Yaskawa INFORM job: hydraulic_planes_program.JBI

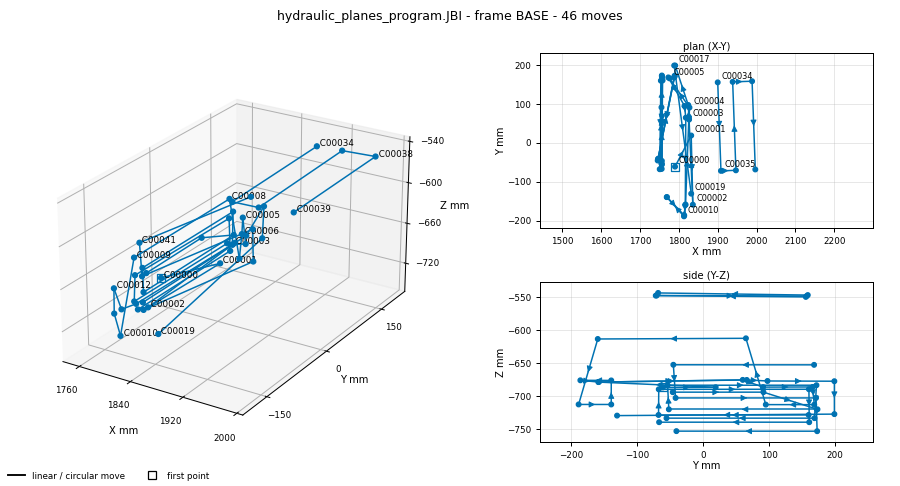
[picture p0: tool path of hydraulic_planes_program.JBI in frame BASE, 46 of 52 moves have a stored position in this frame; points joined in program order, loops and branches not executed]
/JOB
//NAME hydraulic_planes_program
//POS
///NPOS 46,0,46,0,0,0
///TOOL 0
///POSTYPE BASE
///RECTAN
///RCONF 0,0,0,0,0,0,0,0,0,0,0,0,0,0,0,0,0,0,0,0,0,0,0,0
C00000=1790.266260,-61.118146,-686.561623,175.000000,-86.957864,-5.000000
C00001=1831.954921,19.073830,-686.315651,175.000000,-89.878553,-42.967165
C00002=1836.147041,-158.971402,-678.483462,-5.000000,-59.939769,-144.273100
C00003=1826.434318,60.082030,-675.116712,5.000000,-61.318237,147.203233
C00004=1827.467674,91.039273,-686.093792,175.000000,-89.878553,-42.967165
C00005=1776.092305,166.200158,-685.860832,-175.000000,-89.999999,5.000000
C00006=1773.015262,168.636026,-712.737461,175.000000,-86.957864,-5.000000
C00007=1814.783866,95.105126,-712.668296,5.000000,-89.961663,134.868733
C00008=1817.982946,64.939100,-612.030081,175.000000,-59.162706,-36.238815
C00009=1816.677604,-159.909699,-613.050416,175.000000,-59.645373,36.364554
C00010=1813.343123,-188.991701,-712.402389,-175.000000,-89.962495,44.868708
C00011=1768.928091,-139.457958,-712.449114,-175.000000,-89.999999,5.000000
C00012=1769.441453,-139.453159,-675.944419,175.000000,-86.957864,-5.000000
C00013=1813.995933,-186.333152,-675.775252,175.000000,-89.860276,43.447212
C00014=1817.301672,-158.444384,-678.443506,175.000000,-60.142921,35.349719
C00015=1825.978625,66.227215,-675.229416,175.000000,-58.601867,-37.216727
C00016=1824.274715,97.685087,-676.791427,5.000000,-89.849901,133.447578
C00017=1790.762018,199.171368,-677.155686,-175.000000,-89.999999,5.000000
C00018=1788.152021,199.213725,-727.087548,175.000000,-86.957864,-5.000000
C00019=1831.944525,-130.625030,-729.338750,180.000000,-60.000000,0.000000
C00020=1756.349272,-46.141377,-693.754512,5.000000,-89.857180,175.000000
C00021=1755.399155,91.548361,-693.758382,5.000000,-89.857180,175.000000
C00022=1756.387865,173.552879,-719.824458,5.000000,-89.857180,175.000000
C00023=1755.391181,-52.033493,-719.824484,5.000000,-89.857180,175.000000
C00024=1755.768973,-53.986868,-683.221136,5.000000,-89.857180,175.000000
C00025=1756.321618,172.003597,-683.222222,5.000000,-89.857180,175.000000
C00026=1756.861736,169.068743,-733.220999,5.000000,-89.857180,175.000000
C00027=1756.478831,-55.593134,-733.219504,180.000000,-60.000000,0.000000
C00028=1753.816844,160.170606,-728.362357,-5.000000,-87.376565,175.000000
C00029=1750.864769,-67.689122,-728.388394,-5.000000,-87.376565,175.000000
C00030=1752.780642,-67.367991,-689.430064,-5.000000,-87.376565,175.000000
C00031=1756.818776,160.582398,-689.354311,-5.000000,-87.376565,175.000000
C00032=1758.269844,161.023273,-739.340500,-5.000000,-87.376565,175.000000
C00033=1755.987664,-66.800990,-739.335855,180.000000,-60.000000,0.000000
C00034=1900.141403,155.863057,-549.188650,175.000000,-5.000000,5.000000
C00035=1908.499765,-71.912467,-547.251638,175.000000,-5.000000,5.000000
C00036=1946.984303,-70.512261,-547.021638,175.000000,-5.000000,5.000000
C00037=1938.629923,157.154756,-547.865638,175.000000,-5.000000,5.000000
C00038=1988.606888,158.835908,-546.390638,175.000000,-5.000000,5.000000
C00039=1996.941331,-68.287794,-543.165638,175.000000,-5.000000,5.000000
C00040=1787.945105,168.400189,-652.296237,5.000000,-82.585527,-175.000000
C00041=1745.633077,-45.215626,-652.194331,5.000000,-82.585527,-175.000000
C00042=1746.401907,-41.803375,-702.518754,5.000000,-82.585527,-175.000000
C00043=1789.334500,171.346579,-702.527671,5.000000,-82.585527,-175.000000
C00044=1789.323694,173.045553,-753.012360,5.000000,-82.585527,-175.000000
C00045=1746.936745,-40.568483,-752.920252,180.000000,-60.000000,0.000000
///POSTYPE PULSE
///PULSE
EC00000=0.0
EC00001=0.0
EC00002=0.0
EC00003=0.0
EC00004=0.0
EC00005=0.0
EC00006=0.0
EC00007=0.0
EC00008=0.0
EC00009=0.0
EC00010=0.0
EC00011=0.0
EC00012=0.0
EC00013=0.0
EC00014=0.0
EC00015=0.0
EC00016=0.0
EC00017=0.0
EC00018=0.0
EC00019=0.0
EC00020=91136.0
EC00021=91136.0
EC00022=91136.0
EC00023=91136.0
EC00024=91136.0
EC00025=91136.0
EC00026=91136.0
EC00027=91136.0
EC00028=183296.0
EC00029=183296.0
EC00030=183296.0
EC00031=183296.0
EC00032=183296.0
EC00033=183296.0
EC00034=186368.0
EC00035=186368.0
EC00036=186368.0
EC00037=186368.0
EC00038=186368.0
EC00039=186368.0
EC00040=252928.0
EC00041=252928.0
EC00042=252928.0
EC00043=252928.0
EC00044=252928.0
EC00045=252928.0
//INST
///DATE 2023/08/16 16:00
///ATTR SC,RW,RJ
////FRAME BASE
///GROUP1 RB1,ST1
NOP
MOVJ P009 EX000 VJ=15.00
MOVJ C00000 EC00000 VJ=15.0
CALL JOB:SPYON
MOVL C00001 EC00001 V=150.0
MOVL C00002 EC00002 V=150.0
MOVL C00003 EC00003 V=150.0
MOVL C00004 EC00004 V=150.0
MOVL C00005 EC00005 V=150.0
MOVL C00006 EC00006 V=150.0
MOVL C00007 EC00007 V=150.0
MOVL C00008 EC00008 V=150.0
MOVL C00009 EC00009 V=150.0
MOVL C00010 EC00010 V=150.0
MOVL C00011 EC00011 V=150.0
MOVL C00012 EC00012 V=150.0
MOVL C00013 EC00013 V=150.0
MOVL C00014 EC00014 V=150.0
MOVL C00015 EC00015 V=150.0
MOVL C00016 EC00016 V=150.0
MOVL C00017 EC00017 V=150.0
MOVL C00018 EC00018 V=150.0
MOVL C00019 EC00019 V=150.0
CALL JOB:SPYOF
MOVJ P009 VJ=15.00
MOVJ C00020 EC00020 VJ=15.0
CALL JOB:SPYON
MOVL C00021 EC00021 V=150.0
MOVL C00022 EC00022 V=150.0
MOVL C00023 EC00023 V=150.0
MOVL C00024 EC00024 V=150.0
MOVL C00025 EC00025 V=150.0
MOVL C00026 EC00026 V=150.0
MOVL C00027 EC00027 V=150.0
CALL JOB:SPYOF
MOVJ P009 VJ=15.00
MOVJ C00028 EC00028 VJ=15.0
CALL JOB:SPYON
MOVL C00029 EC00029 V=150.0
MOVL C00030 EC00030 V=150.0
MOVL C00031 EC00031 V=150.0
MOVL C00032 EC00032 V=150.0
MOVL C00033 EC00033 V=150.0
CALL JOB:SPYOF
MOVJ P009 VJ=15.00
MOVJ C00034 EC00034 VJ=15.0
CALL JOB:SPYON
MOVL C00035 EC00035 V=150.0
MOVL C00036 EC00036 V=150.0
MOVL C00037 EC00037 V=150.0
MOVL C00038 EC00038 V=150.0
MOVL C00039 EC00039 V=150.0
CALL JOB:SPYOF
MOVJ P009 VJ=15.00
MOVJ C00040 EC00040 VJ=15.0
CALL JOB:SPYON
MOVL C00041 EC00041 V=150.0
MOVL C00042 EC00042 V=150.0
MOVL C00043 EC00043 V=150.0
MOVL C00044 EC00044 V=150.0
MOVL C00045 EC00045 V=150.0
CALL JOB:SPYOF
MOVJ P009 VJ=15.00
END
